(* Logix 5000 project; controller Sucrose_Main Emulate 5570 rev 20.12; software revision 20.01; part 22 of 30 *)
(* tags used below, declared in another part *)
   ONESHOTBITS : INT[10];
   Rung_Comment : BOOL;
   SucroseFiltration : Area_Program;
(* Master_Main, continued *)

ROUTINE HMI_old   (* ladder *)
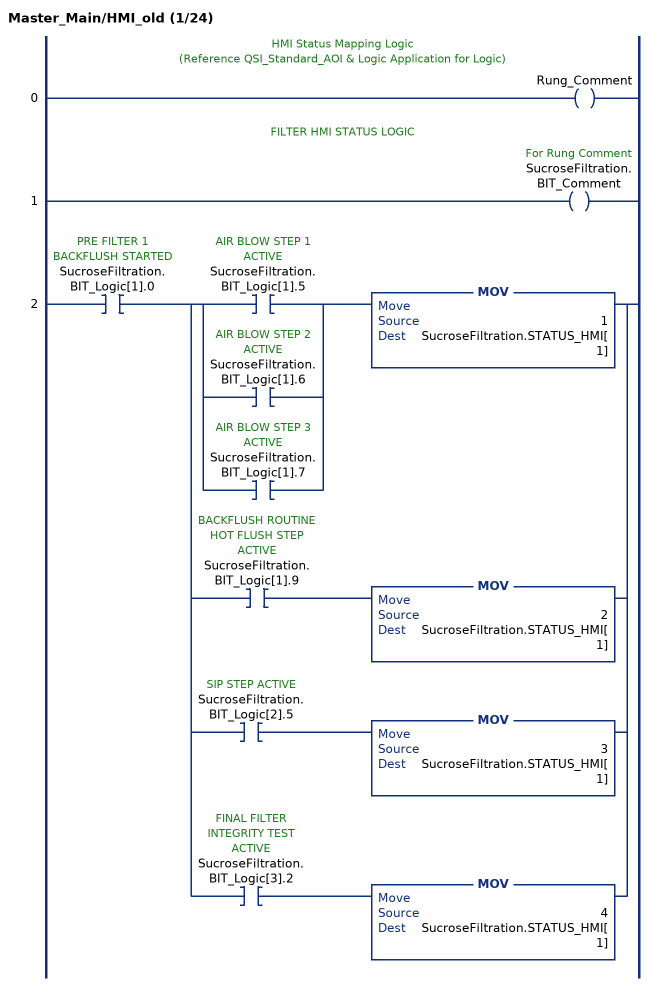
   // HMI Status Mapping Logic
   // (Reference QSI_Standard_AOI & Logic Application for Logic)
   0: OTE(Rung_Comment);
   // FILTER HMI STATUS LOGIC
   1: OTE(SucroseFiltration.BIT_Comment);
   2: XIC(SucroseFiltration.BIT_Logic[1].0)[[XIC(SucroseFiltration.BIT_Logic[1].5) ,XIC(SucroseFiltration.BIT_Logic[1].6) ,XIC(SucroseFiltration.BIT_Logic[1].7) ] MOV(1,SucroseFiltration.STATUS_HMI[1]) ,XIC(SucroseFiltration.BIT_Logic[1].9) MOV(2,SucroseFiltration.STATUS_HMI[1]) ,XIC(SucroseFiltration.BIT_Logic[2].5) MOV(3,SucroseFiltration.STATUS_HMI[1]) ,XIC(SucroseFiltration.BIT_Logic[3].2) MOV(4,SucroseFiltration.STATUS_HMI[1]) ];
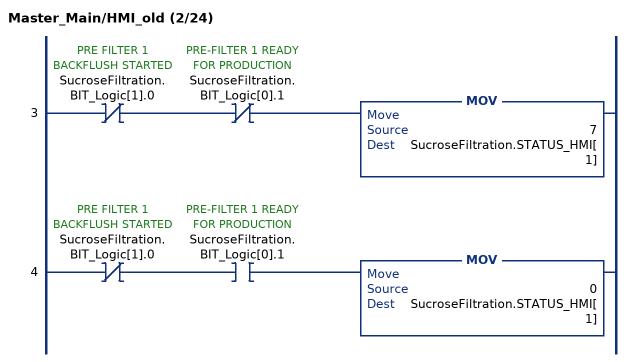
   3: XIO(SucroseFiltration.BIT_Logic[1].0)XIO(SucroseFiltration.BIT_Logic[0].1)MOV(7,SucroseFiltration.STATUS_HMI[1]);
   4: XIO(SucroseFiltration.BIT_Logic[1].0)XIC(SucroseFiltration.BIT_Logic[0].1)MOV(0,SucroseFiltration.STATUS_HMI[1]);
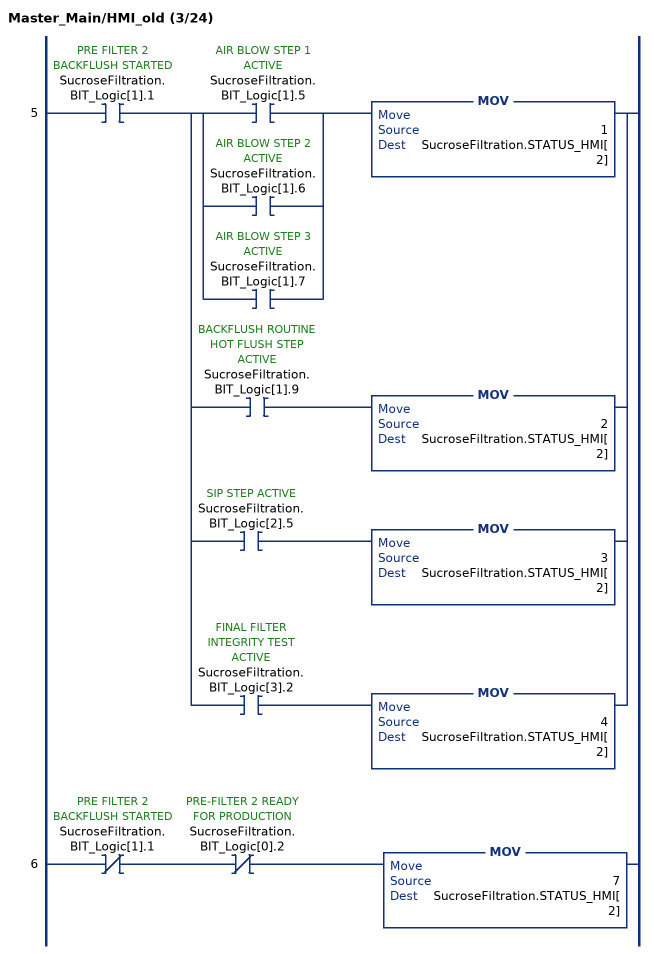
   5: XIC(SucroseFiltration.BIT_Logic[1].1)[[XIC(SucroseFiltration.BIT_Logic[1].5) ,XIC(SucroseFiltration.BIT_Logic[1].6) ,XIC(SucroseFiltration.BIT_Logic[1].7) ] MOV(1,SucroseFiltration.STATUS_HMI[2]) ,XIC(SucroseFiltration.BIT_Logic[1].9) MOV(2,SucroseFiltration.STATUS_HMI[2]) ,XIC(SucroseFiltration.BIT_Logic[2].5) MOV(3,SucroseFiltration.STATUS_HMI[2]) ,XIC(SucroseFiltration.BIT_Logic[3].2) MOV(4,SucroseFiltration.STATUS_HMI[2]) ];
   6: XIO(SucroseFiltration.BIT_Logic[1].1)XIO(SucroseFiltration.BIT_Logic[0].2)MOV(7,SucroseFiltration.STATUS_HMI[2]);
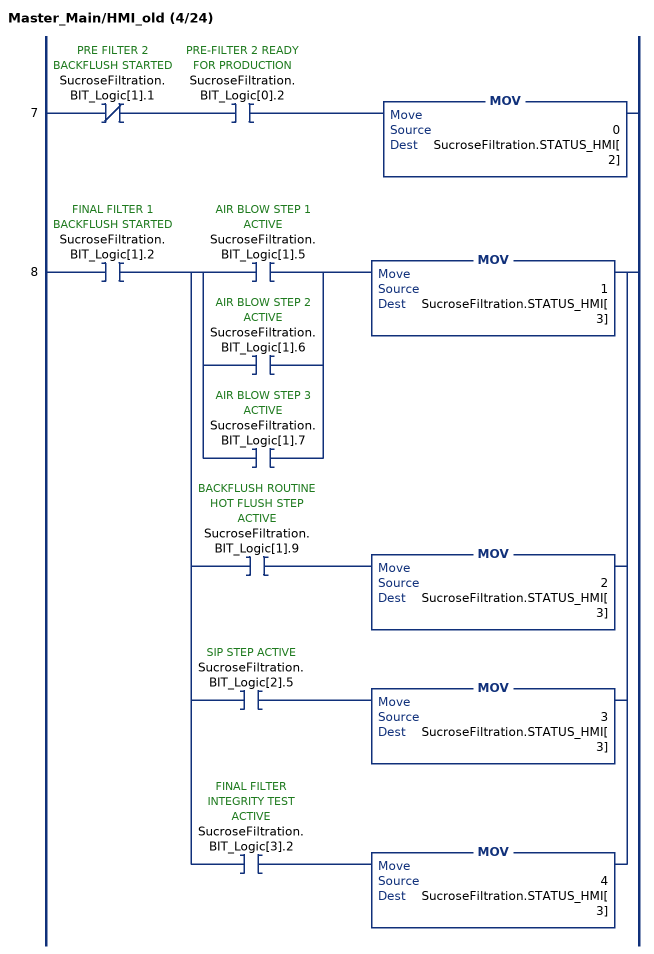
   7: XIO(SucroseFiltration.BIT_Logic[1].1)XIC(SucroseFiltration.BIT_Logic[0].2)MOV(0,SucroseFiltration.STATUS_HMI[2]);
   8: XIC(SucroseFiltration.BIT_Logic[1].2)[[XIC(SucroseFiltration.BIT_Logic[1].5) ,XIC(SucroseFiltration.BIT_Logic[1].6) ,XIC(SucroseFiltration.BIT_Logic[1].7) ] MOV(1,SucroseFiltration.STATUS_HMI[3]) ,XIC(SucroseFiltration.BIT_Logic[1].9) MOV(2,SucroseFiltration.STATUS_HMI[3]) ,XIC(SucroseFiltration.BIT_Logic[2].5) MOV(3,SucroseFiltration.STATUS_HMI[3]) ,XIC(SucroseFiltration.BIT_Logic[3].2) MOV(4,SucroseFiltration.STATUS_HMI[3]) ];
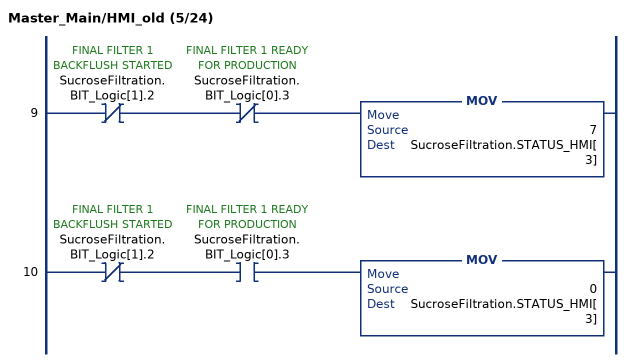
   9: XIO(SucroseFiltration.BIT_Logic[1].2)XIO(SucroseFiltration.BIT_Logic[0].3)MOV(7,SucroseFiltration.STATUS_HMI[3]);
   10: XIO(SucroseFiltration.BIT_Logic[1].2)XIC(SucroseFiltration.BIT_Logic[0].3)MOV(0,SucroseFiltration.STATUS_HMI[3]);
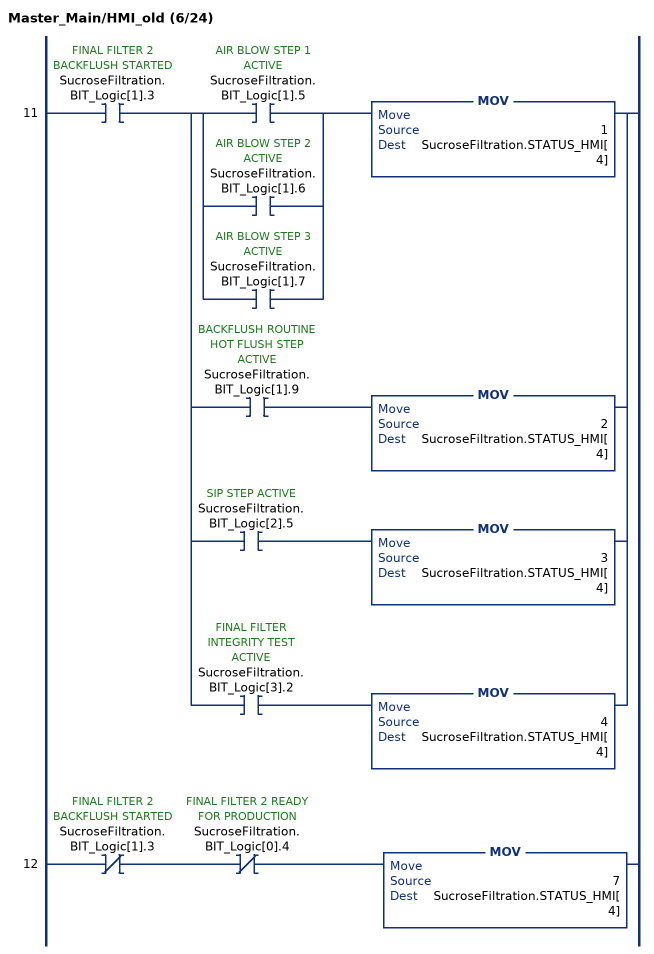
   11: XIC(SucroseFiltration.BIT_Logic[1].3)[[XIC(SucroseFiltration.BIT_Logic[1].5) ,XIC(SucroseFiltration.BIT_Logic[1].6) ,XIC(SucroseFiltration.BIT_Logic[1].7) ] MOV(1,SucroseFiltration.STATUS_HMI[4]) ,XIC(SucroseFiltration.BIT_Logic[1].9) MOV(2,SucroseFiltration.STATUS_HMI[4]) ,XIC(SucroseFiltration.BIT_Logic[2].5) MOV(3,SucroseFiltration.STATUS_HMI[4]) ,XIC(SucroseFiltration.BIT_Logic[3].2) MOV(4,SucroseFiltration.STATUS_HMI[4]) ];
   12: XIO(SucroseFiltration.BIT_Logic[1].3)XIO(SucroseFiltration.BIT_Logic[0].4)MOV(7,SucroseFiltration.STATUS_HMI[4]);
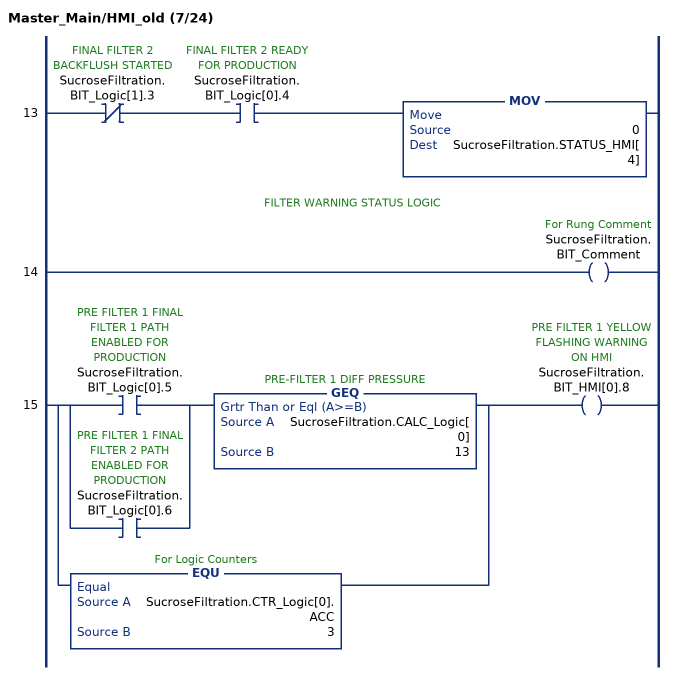
   13: XIO(SucroseFiltration.BIT_Logic[1].3)XIC(SucroseFiltration.BIT_Logic[0].4)MOV(0,SucroseFiltration.STATUS_HMI[4]);
   // FILTER WARNING STATUS LOGIC
   14: OTE(SucroseFiltration.BIT_Comment);
   15: [[XIC(SucroseFiltration.BIT_Logic[0].5) ,XIC(SucroseFiltration.BIT_Logic[0].6) ] GEQ(SucroseFiltration.CALC_Logic[0],13) ,EQU(SucroseFiltration.CTR_Logic[0].ACC,3) ]OTE(SucroseFiltration.BIT_HMI[0].8);
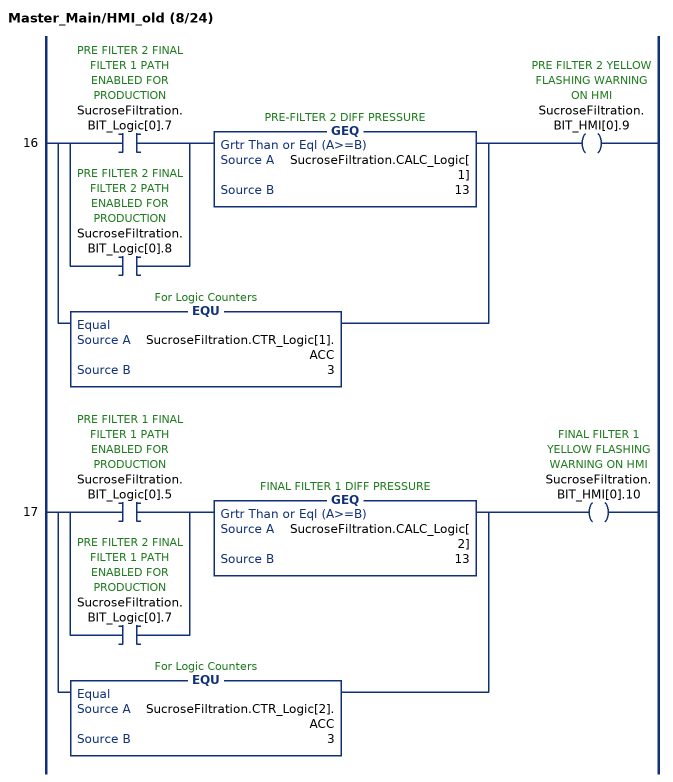
   16: [[XIC(SucroseFiltration.BIT_Logic[0].7) ,XIC(SucroseFiltration.BIT_Logic[0].8) ] GEQ(SucroseFiltration.CALC_Logic[1],13) ,EQU(SucroseFiltration.CTR_Logic[1].ACC,3) ]OTE(SucroseFiltration.BIT_HMI[0].9);
   17: [[XIC(SucroseFiltration.BIT_Logic[0].5) ,XIC(SucroseFiltration.BIT_Logic[0].7) ] GEQ(SucroseFiltration.CALC_Logic[2],13) ,EQU(SucroseFiltration.CTR_Logic[2].ACC,3) ]OTE(SucroseFiltration.BIT_HMI[0].10);
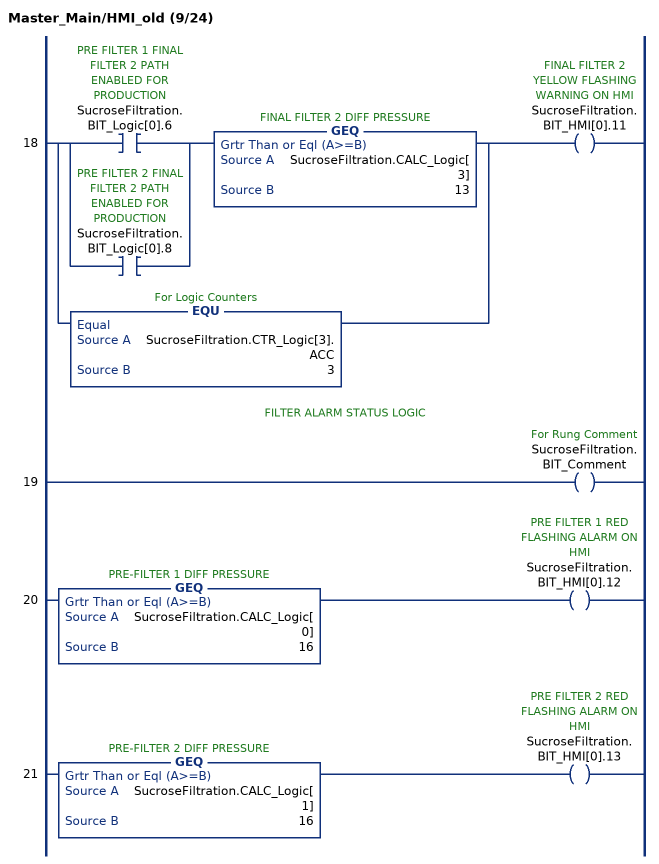
   18: [[XIC(SucroseFiltration.BIT_Logic[0].6) ,XIC(SucroseFiltration.BIT_Logic[0].8) ] GEQ(SucroseFiltration.CALC_Logic[3],13) ,EQU(SucroseFiltration.CTR_Logic[3].ACC,3) ]OTE(SucroseFiltration.BIT_HMI[0].11);
   // FILTER ALARM STATUS LOGIC
   19: OTE(SucroseFiltration.BIT_Comment);
   20: GEQ(SucroseFiltration.CALC_Logic[0],16)OTE(SucroseFiltration.BIT_HMI[0].12);
   21: GEQ(SucroseFiltration.CALC_Logic[1],16)OTE(SucroseFiltration.BIT_HMI[0].13);
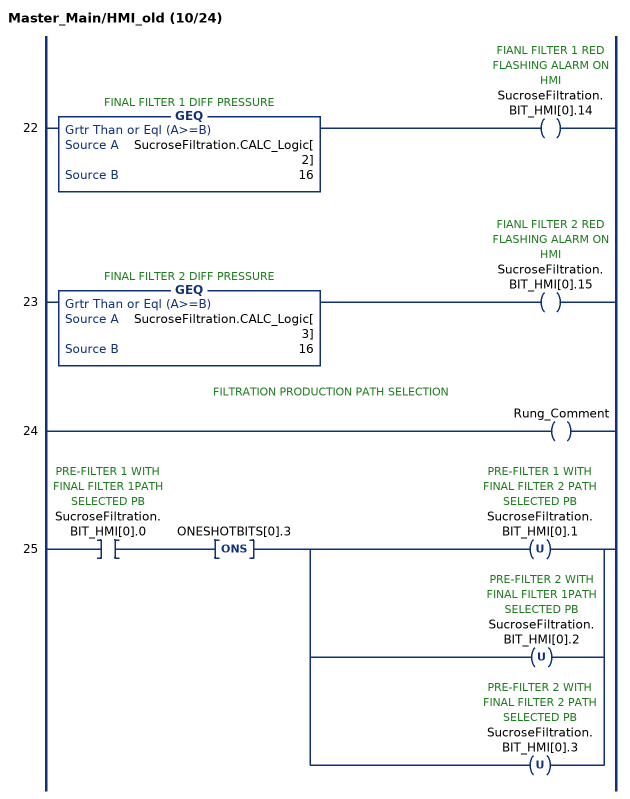
   22: GEQ(SucroseFiltration.CALC_Logic[2],16)OTE(SucroseFiltration.BIT_HMI[0].14);
   23: GEQ(SucroseFiltration.CALC_Logic[3],16)OTE(SucroseFiltration.BIT_HMI[0].15);
   // FILTRATION PRODUCTION PATH SELECTION
   24: OTE(Rung_Comment);
   25: XIC(SucroseFiltration.BIT_HMI[0].0)ONS(ONESHOTBITS[0].3)[OTU(SucroseFiltration.BIT_HMI[0].1) ,OTU(SucroseFiltration.BIT_HMI[0].2) ,OTU(SucroseFiltration.BIT_HMI[0].3) ];
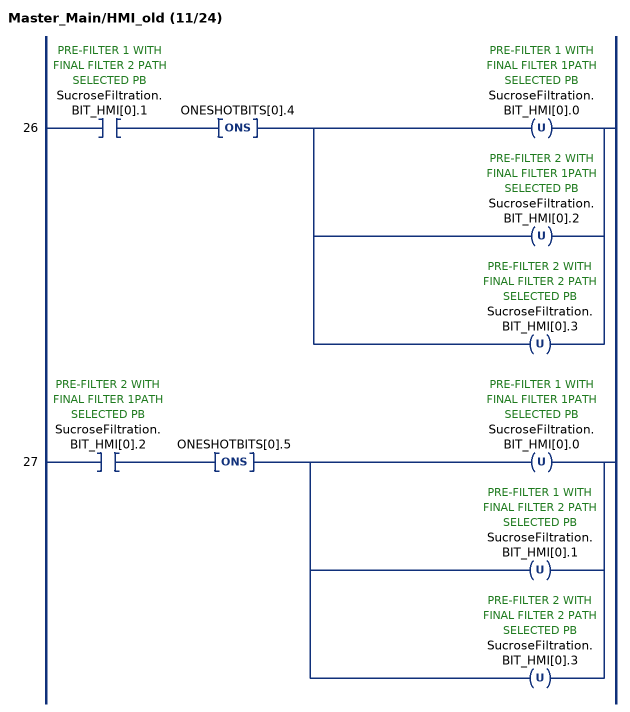
   26: XIC(SucroseFiltration.BIT_HMI[0].1)ONS(ONESHOTBITS[0].4)[OTU(SucroseFiltration.BIT_HMI[0].0) ,OTU(SucroseFiltration.BIT_HMI[0].2) ,OTU(SucroseFiltration.BIT_HMI[0].3) ];
   27: XIC(SucroseFiltration.BIT_HMI[0].2)ONS(ONESHOTBITS[0].5)[OTU(SucroseFiltration.BIT_HMI[0].0) ,OTU(SucroseFiltration.BIT_HMI[0].1) ,OTU(SucroseFiltration.BIT_HMI[0].3) ];
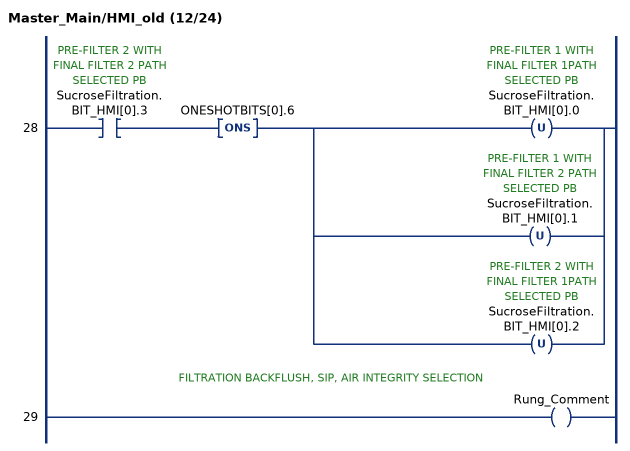
   28: XIC(SucroseFiltration.BIT_HMI[0].3)ONS(ONESHOTBITS[0].6)[OTU(SucroseFiltration.BIT_HMI[0].0) ,OTU(SucroseFiltration.BIT_HMI[0].1) ,OTU(SucroseFiltration.BIT_HMI[0].2) ];
   // FILTRATION BACKFLUSH, SIP, AIR INTEGRITY SELECTION
   29: OTE(Rung_Comment);
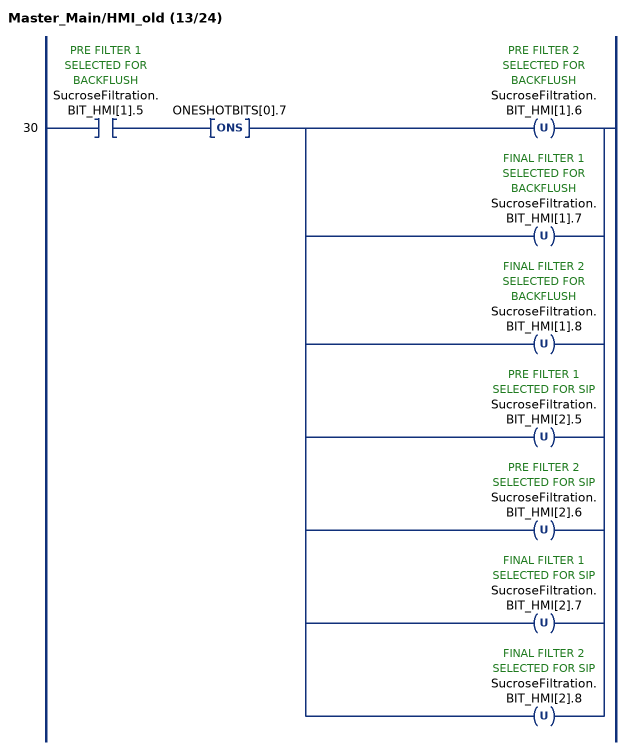
   30: XIC(SucroseFiltration.BIT_HMI[1].5)ONS(ONESHOTBITS[0].7)[OTU(SucroseFiltration.BIT_HMI[1].6) ,OTU(SucroseFiltration.BIT_HMI[1].7) ,OTU(SucroseFiltration.BIT_HMI[1].8) ,OTU(SucroseFiltration.BIT_HMI[2].5) ,OTU(SucroseFiltration.BIT_HMI[2].6) ,OTU(SucroseFiltration.BIT_HMI[2].7) ,OTU(SucroseFiltration.BIT_HMI[2].8) ];
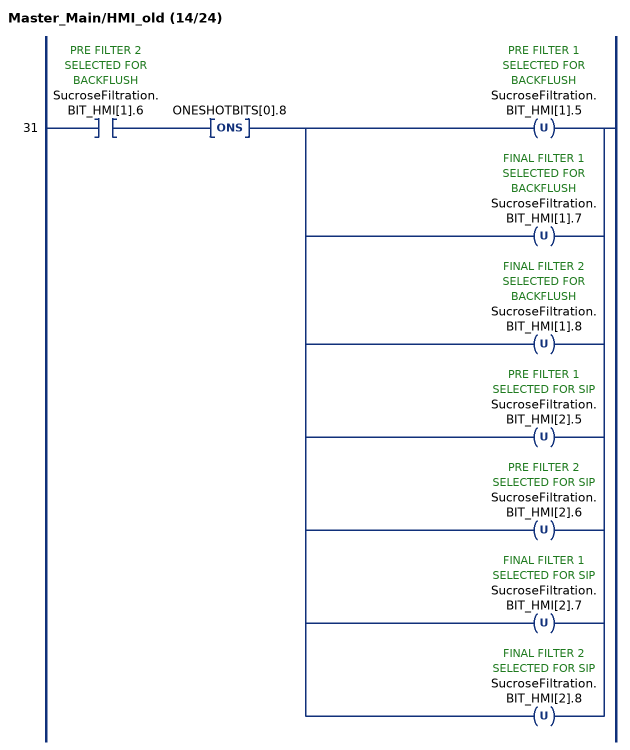
   31: XIC(SucroseFiltration.BIT_HMI[1].6)ONS(ONESHOTBITS[0].8)[OTU(SucroseFiltration.BIT_HMI[1].5) ,OTU(SucroseFiltration.BIT_HMI[1].7) ,OTU(SucroseFiltration.BIT_HMI[1].8) ,OTU(SucroseFiltration.BIT_HMI[2].5) ,OTU(SucroseFiltration.BIT_HMI[2].6) ,OTU(SucroseFiltration.BIT_HMI[2].7) ,OTU(SucroseFiltration.BIT_HMI[2].8) ];
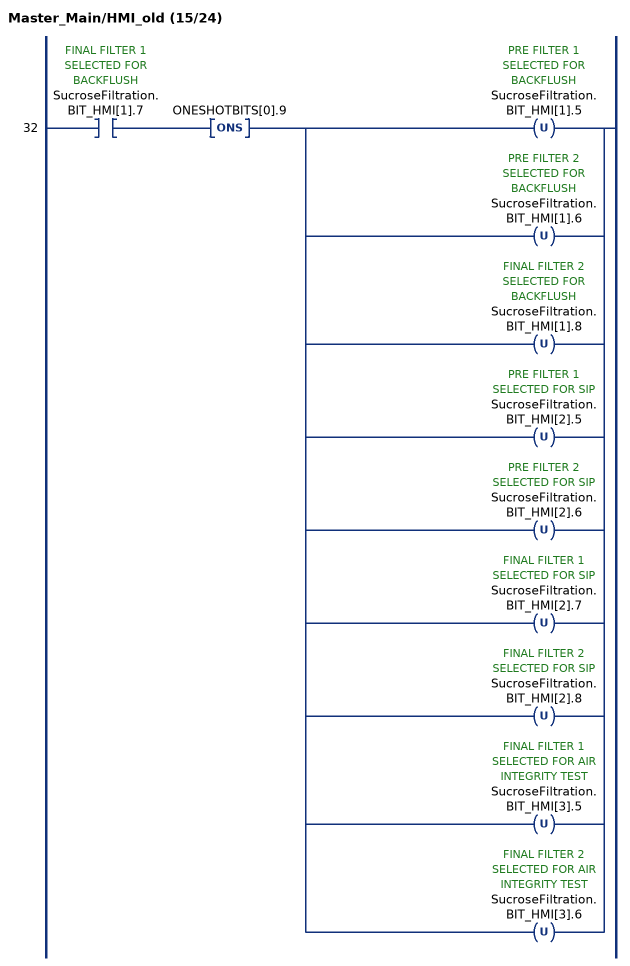
   32: XIC(SucroseFiltration.BIT_HMI[1].7)ONS(ONESHOTBITS[0].9)[OTU(SucroseFiltration.BIT_HMI[1].5) ,OTU(SucroseFiltration.BIT_HMI[1].6) ,OTU(SucroseFiltration.BIT_HMI[1].8) ,OTU(SucroseFiltration.BIT_HMI[2].5) ,OTU(SucroseFiltration.BIT_HMI[2].6) ,OTU(SucroseFiltration.BIT_HMI[2].7) ,OTU(SucroseFiltration.BIT_HMI[2].8) ,OTU(SucroseFiltration.BIT_HMI[3].5) ,OTU(SucroseFiltration.BIT_HMI[3].6) ];
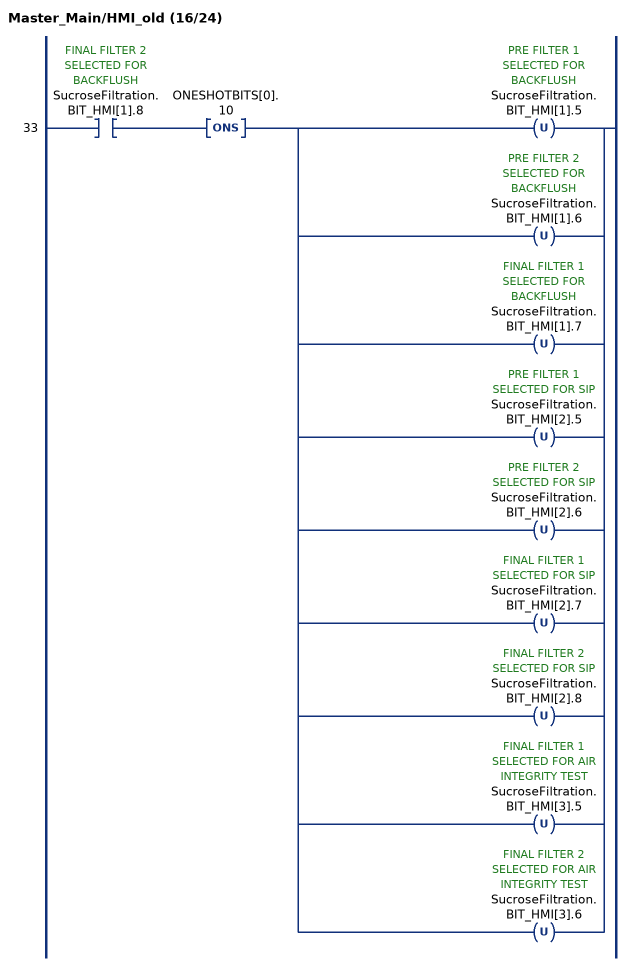
   33: XIC(SucroseFiltration.BIT_HMI[1].8)ONS(ONESHOTBITS[0].10)[OTU(SucroseFiltration.BIT_HMI[1].5) ,OTU(SucroseFiltration.BIT_HMI[1].6) ,OTU(SucroseFiltration.BIT_HMI[1].7) ,OTU(SucroseFiltration.BIT_HMI[2].5) ,OTU(SucroseFiltration.BIT_HMI[2].6) ,OTU(SucroseFiltration.BIT_HMI[2].7) ,OTU(SucroseFiltration.BIT_HMI[2].8) ,OTU(SucroseFiltration.BIT_HMI[3].5) ,OTU(SucroseFiltration.BIT_HMI[3].6) ];
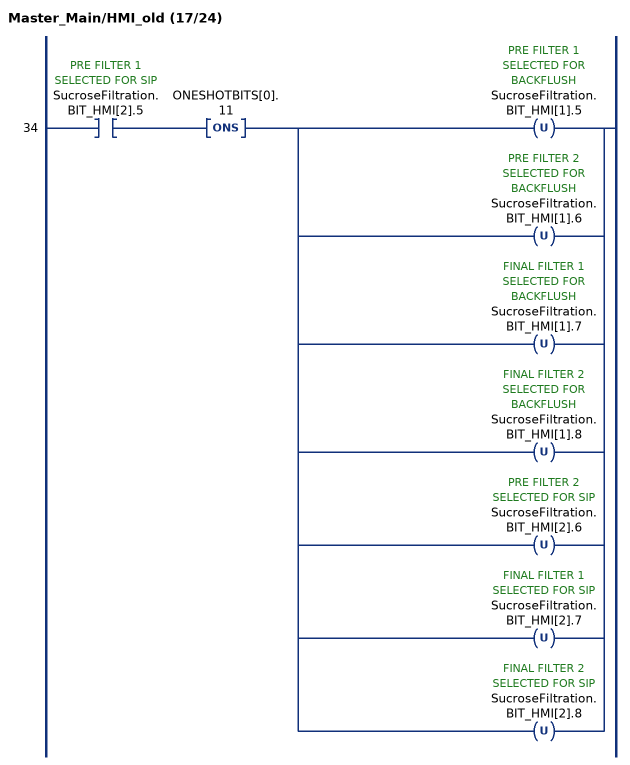
   34: XIC(SucroseFiltration.BIT_HMI[2].5)ONS(ONESHOTBITS[0].11)[OTU(SucroseFiltration.BIT_HMI[1].5) ,OTU(SucroseFiltration.BIT_HMI[1].6) ,OTU(SucroseFiltration.BIT_HMI[1].7) ,OTU(SucroseFiltration.BIT_HMI[1].8) ,OTU(SucroseFiltration.BIT_HMI[2].6) ,OTU(SucroseFiltration.BIT_HMI[2].7) ,OTU(SucroseFiltration.BIT_HMI[2].8) ];
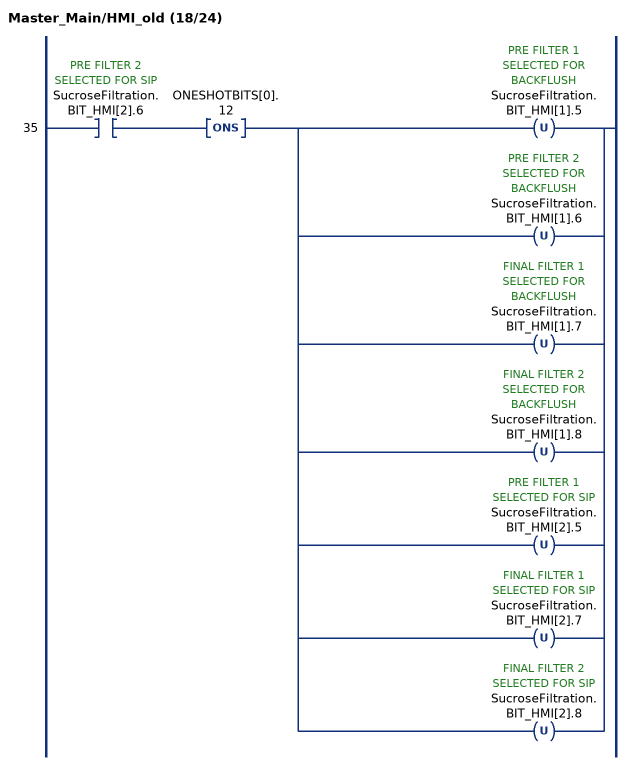
   35: XIC(SucroseFiltration.BIT_HMI[2].6)ONS(ONESHOTBITS[0].12)[OTU(SucroseFiltration.BIT_HMI[1].5) ,OTU(SucroseFiltration.BIT_HMI[1].6) ,OTU(SucroseFiltration.BIT_HMI[1].7) ,OTU(SucroseFiltration.BIT_HMI[1].8) ,OTU(SucroseFiltration.BIT_HMI[2].5) ,OTU(SucroseFiltration.BIT_HMI[2].7) ,OTU(SucroseFiltration.BIT_HMI[2].8) ];
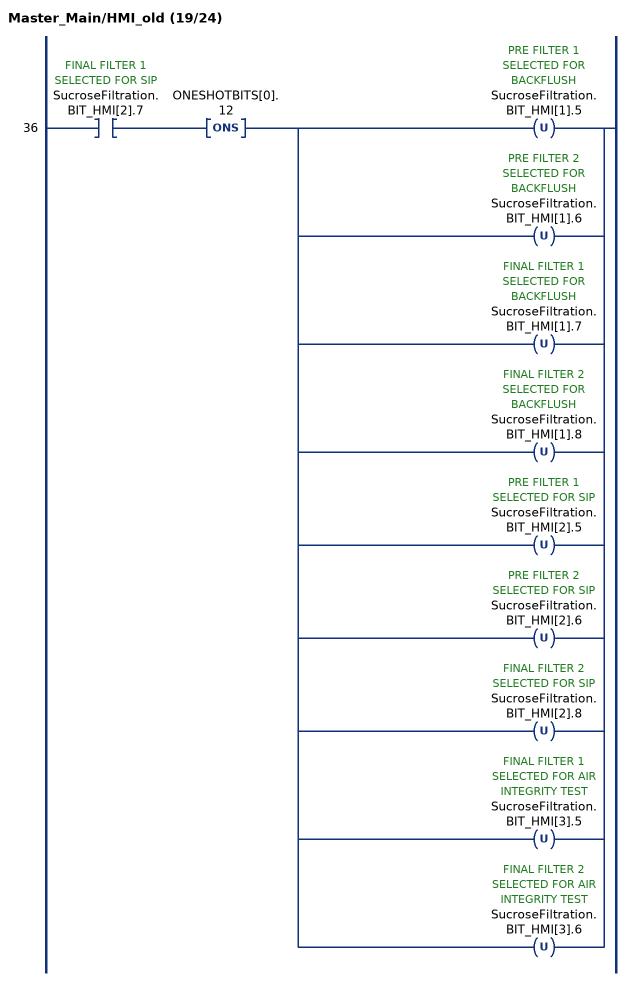
   36: XIC(SucroseFiltration.BIT_HMI[2].7)ONS(ONESHOTBITS[0].12)[OTU(SucroseFiltration.BIT_HMI[1].5) ,OTU(SucroseFiltration.BIT_HMI[1].6) ,OTU(SucroseFiltration.BIT_HMI[1].7) ,OTU(SucroseFiltration.BIT_HMI[1].8) ,OTU(SucroseFiltration.BIT_HMI[2].5) ,OTU(SucroseFiltration.BIT_HMI[2].6) ,OTU(SucroseFiltration.BIT_HMI[2].8) ,OTU(SucroseFiltration.BIT_HMI[3].5) ,OTU(SucroseFiltration.BIT_HMI[3].6) ];
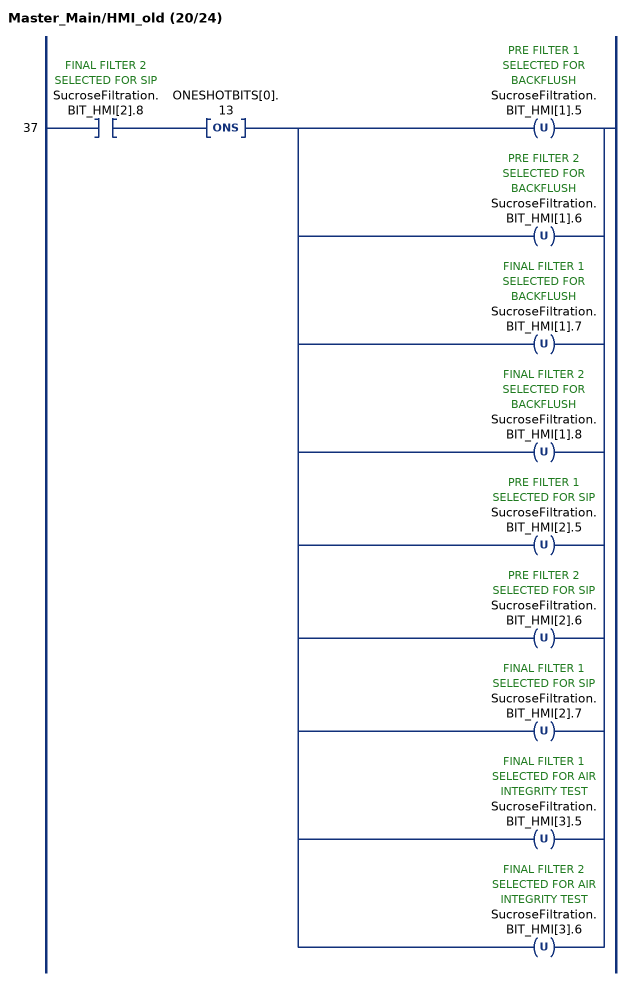
   37: XIC(SucroseFiltration.BIT_HMI[2].8)ONS(ONESHOTBITS[0].13)[OTU(SucroseFiltration.BIT_HMI[1].5) ,OTU(SucroseFiltration.BIT_HMI[1].6) ,OTU(SucroseFiltration.BIT_HMI[1].7) ,OTU(SucroseFiltration.BIT_HMI[1].8) ,OTU(SucroseFiltration.BIT_HMI[2].5) ,OTU(SucroseFiltration.BIT_HMI[2].6) ,OTU(SucroseFiltration.BIT_HMI[2].7) ,OTU(SucroseFiltration.BIT_HMI[3].5) ,OTU(SucroseFiltration.BIT_HMI[3].6) ];
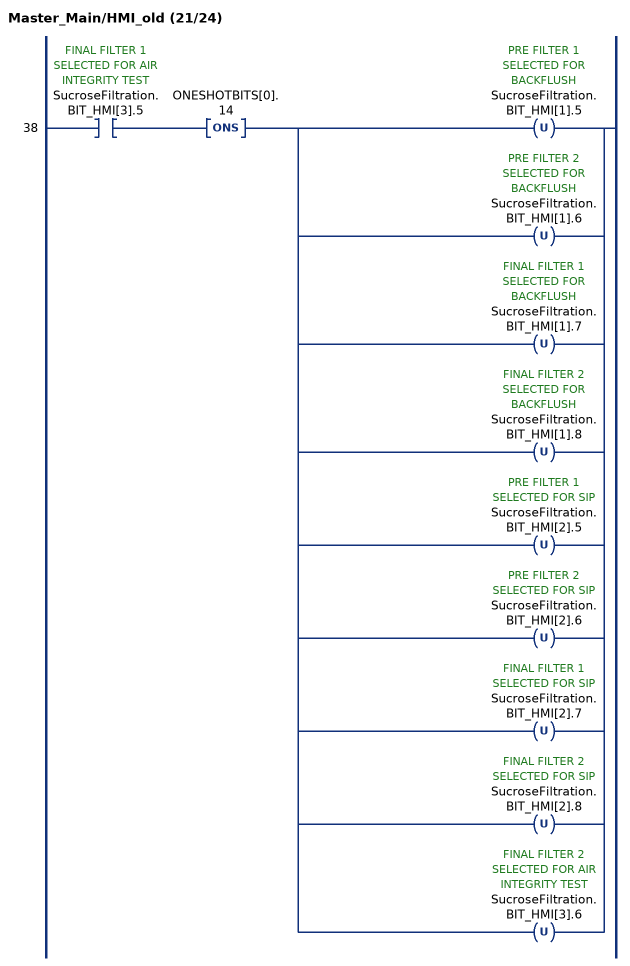
   38: XIC(SucroseFiltration.BIT_HMI[3].5)ONS(ONESHOTBITS[0].14)[OTU(SucroseFiltration.BIT_HMI[1].5) ,OTU(SucroseFiltration.BIT_HMI[1].6) ,OTU(SucroseFiltration.BIT_HMI[1].7) ,OTU(SucroseFiltration.BIT_HMI[1].8) ,OTU(SucroseFiltration.BIT_HMI[2].5) ,OTU(SucroseFiltration.BIT_HMI[2].6) ,OTU(SucroseFiltration.BIT_HMI[2].7) ,OTU(SucroseFiltration.BIT_HMI[2].8) ,OTU(SucroseFiltration.BIT_HMI[3].6) ];
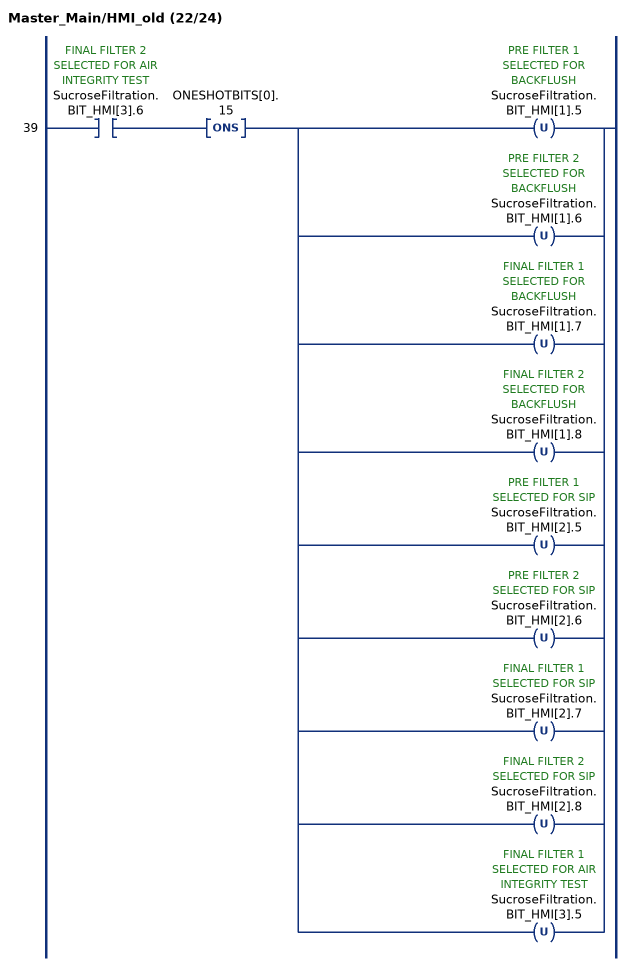
   39: XIC(SucroseFiltration.BIT_HMI[3].6)ONS(ONESHOTBITS[0].15)[OTU(SucroseFiltration.BIT_HMI[1].5) ,OTU(SucroseFiltration.BIT_HMI[1].6) ,OTU(SucroseFiltration.BIT_HMI[1].7) ,OTU(SucroseFiltration.BIT_HMI[1].8) ,OTU(SucroseFiltration.BIT_HMI[2].5) ,OTU(SucroseFiltration.BIT_HMI[2].6) ,OTU(SucroseFiltration.BIT_HMI[2].7) ,OTU(SucroseFiltration.BIT_HMI[2].8) ,OTU(SucroseFiltration.BIT_HMI[3].5) ];
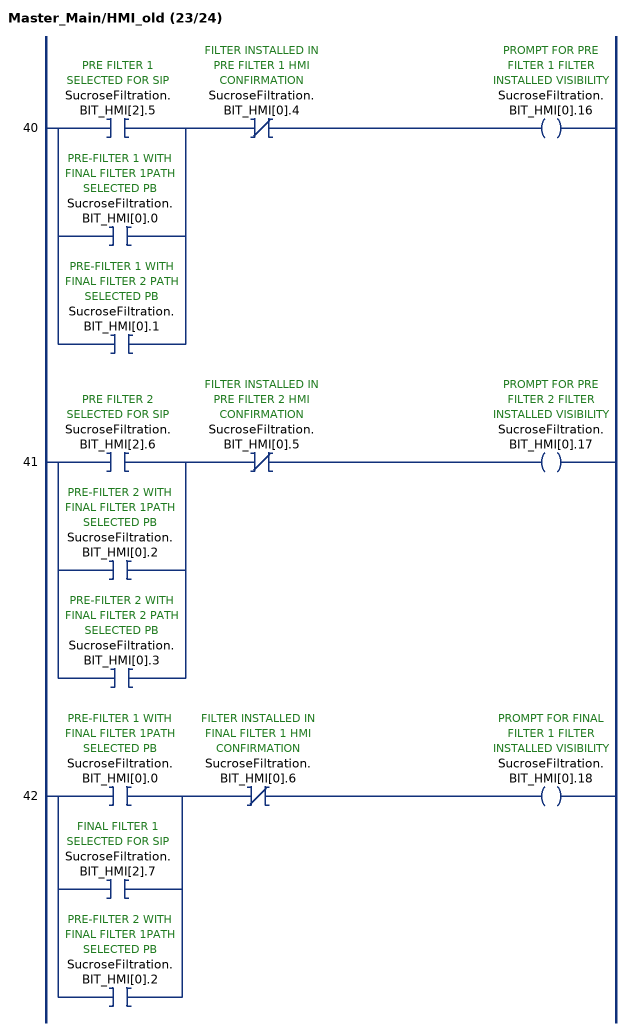
   40: [XIC(SucroseFiltration.BIT_HMI[2].5) ,XIC(SucroseFiltration.BIT_HMI[0].0) ,XIC(SucroseFiltration.BIT_HMI[0].1) ]XIO(SucroseFiltration.BIT_HMI[0].4)OTE(SucroseFiltration.BIT_HMI[0].16);
   41: [XIC(SucroseFiltration.BIT_HMI[2].6) ,XIC(SucroseFiltration.BIT_HMI[0].2) ,XIC(SucroseFiltration.BIT_HMI[0].3) ]XIO(SucroseFiltration.BIT_HMI[0].5)OTE(SucroseFiltration.BIT_HMI[0].17);
   42: [XIC(SucroseFiltration.BIT_HMI[0].0) ,XIC(SucroseFiltration.BIT_HMI[2].7) ,XIC(SucroseFiltration.BIT_HMI[0].2) ]XIO(SucroseFiltration.BIT_HMI[0].6)OTE(SucroseFiltration.BIT_HMI[0].18);
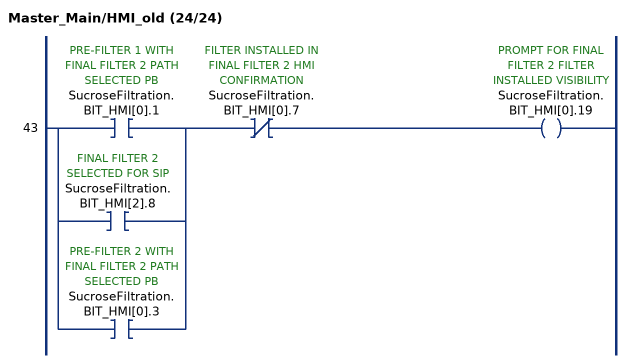
   43: [XIC(SucroseFiltration.BIT_HMI[0].1) ,XIC(SucroseFiltration.BIT_HMI[2].8) ,XIC(SucroseFiltration.BIT_HMI[0].3) ]XIO(SucroseFiltration.BIT_HMI[0].7)OTE(SucroseFiltration.BIT_HMI[0].19);
END_ROUTINE
